(* PLC project RTC_PulseGen_TwinForge, TwinForge TwinForge 0.1.0 *)
(* stored: creationDateTime 2026-07-26T05:06:13.190491+00:00 *)

PROGRAM PLC_PRG
  VAR
    fbRTC_PulseGen : RTC_PulseGen;
    xEnableIn : BOOL := TRUE;
    xEnableOut : BOOL;
    xInp_Enable : BOOL := FALSE;
    diInp_Interval : DINT := 1000;
    xSts_Enabled : BOOL := FALSE;
    xOut : BOOL := FALSE;
  END_VAR

                  fbRTC_PulseGen(
    EnableIn := xEnableIn,
    EnableOut => xEnableOut,
    Inp_Enable := xInp_Enable,
    Inp_Interval := diInp_Interval,
    Sts_Enabled => xSts_Enabled,
    Out => xOut
);
                
END_PROGRAM

FUNCTION_BLOCK RTC_PulseGen
  VAR_INPUT
    EnableIn : BOOL;
    Inp_Enable : BOOL;
    Inp_Interval : DINT;
  END_VAR
  VAR_OUTPUT
    EnableOut : BOOL;
    Sts_Enabled : BOOL;
    Out : BOOL;
  END_VAR
  VAR
    OSR : BOOL;
    TStart : LINT;
    TNow : LINT;
    tfWallClockMilliseconds : SysTime;
    tfWallClockResult : SysTypes.RTS_IEC_RESULT;
  END_VAR

                  EnableOut := EnableIn;
IF EnableIn THEN
    tfWallClockResult := SysTimeRtcHighResGet(tfWallClockMilliseconds);
    IF tfWallClockResult = 0 THEN
        TNow := ULINT_TO_LINT(tfWallClockMilliseconds * ULINT#1000);
    END_IF;
    IF (tfWallClockResult = 0) THEN
        IF ((Inp_Enable AND NOT (OSR)) OR Out) THEN
            TStart := TNow;
        END_IF;
        OSR := Inp_Enable;
        Sts_Enabled := Inp_Enable;
        Out := (Inp_Enable AND ((TNow - TStart) >= (Inp_Interval * 1000)));
    ELSE
        Sts_Enabled := FALSE;
        Out := FALSE;
    END_IF;
END_IF;
                

METHOD FB_Init : BOOL
  VAR_INPUT
    bInitRetains : BOOL;
    bInCopyCode : BOOL;
  END_VAR
                        OSR := 0;
Out := 0;
FB_Init := TRUE;
                      
END_METHOD
END_FUNCTION_BLOCK

CONFIGURATION Application
  RESOURCE Application ON PLC
    TASK MainTask(INTERVAL := T#20ms, PRIORITY := 1);
    PROGRAM PLC_PRG WITH MainTask : PLC_PRG;
  END_RESOURCE
END_CONFIGURATION
